TYPE ST_VIx2000_Pulse :
STRUCT
	nTimestamp 		: T_DCTIME64;
	nFlashDelay 	: UINT;
END_STRUCT
END_TYPE

(* stored: Version 1.1.0.1, ProductVersion 3.1.4024.12
   DUT ST_VIx2000_Pulse: Id {086025bb-7216-455a-b0cf-3fdd6708c858} *)
